FUNCTION_BLOCK FB_TestSuite_CFC EXTENDS TcUnit.FB_TestSuite
VAR_INPUT
END_VAR
VAR_OUTPUT
END_VAR
VAR
END_VAR

END_FUNCTION_BLOCK

(* stored: Version 1.1.0.1, ProductVersion 3.1.4024.12
   POU FB_TestSuite_CFC: Id {a23010cd-0a03-4427-b7d5-a31f1cf67c5e}, SpecialFunc None *)
